TYPE ST_CFG_ProfileRule :
STRUCT
	TU_Type					: INT;
	ReportValue				: INT;
	Minimum					: INT;
	Maximum					: INT;
	Default					: INT;	
END_STRUCT
END_TYPE

(* stored: Version 1.1.0.1, ProductVersion 3.1.4020.6
   DUT ST_CFG_ProfileRule: Id {76e9d1a5-97c2-4982-acf6-88a07558d6c4} *)
